{attribute 'linkalways'} 
{attribute 'no_explicit_call' := 'This FB is a CLASS and must be accessed using methods or properties'}
{attribute 'enable_dynamic_creation'}
FUNCTION_BLOCK Node_F_VN_PutText EXTENDS Node
VAR
    sText : _STRING('');
    ipDestImage : _ITcVnImage;
    nX : _UDINT(1);
    nY : _UDINT(1);
    eFontType : _ETcVnFontType(ETcVnFontType.TCVN_FT_HERSHEY_SIMPLEX);
    fFontScale : _LREAL(1.0);
    //aColor : _TcVnVector4_LREAL;
    hrPrev : _HRESULT(S_OK);
	hresult : _HRESULT(S_OK);
END_VAR

METHOD PUBLIC  Clone : I_Node
VAR
	pNode : POINTER TO Node_F_VN_PutText;
END_VAR
pNode := __NEW(Node_F_VN_PutText);
Clone := pNode^;
END_METHOD

METHOD FB_init : BOOL
VAR_INPUT
	bInitRetains : BOOL; // if TRUE, the retain variables are initialized (warm start / cold start)
	bInCopyCode : BOOL;  // if TRUE, the instance afterwards gets moved into the copy code (online change)
END_VAR
AddInput('sText', sText);
AddInput('ipDestImage', ipDestImage);
//AddInput('aColor', aColor);
AddInput('hrPrev', hrPrev);
AddOutput('ipDestImage', ipDestImage);
AddOutput('hresult',hresult);
AddParameter('nX', nX);
AddParameter('nY', nY);
AddParameter('eFontType', eFontType);
AddParameter('fFontScale', fFontScale);
END_METHOD

METHOD PROTECTED  OnExecute : HRESULT

//REMOVE
VAR
    aColor_Green : TcVnVector4_LREAL := [0, 255, 0];
END_VAR
hresult.Value := F_VN_PutText(
    sText := sText.Value,
	ipDestImage := ipDestImage.Value,
	nX:= nX.Value,
	nY:= nY.Value,
    eFontType := eFontType.Value,
    fFontScale := fFontScale.Value,
    //aColor := aColor.Value,
    aColor := aColor_Green,
	hrPrev:= hrPrev.Value);
END_METHOD

END_FUNCTION_BLOCK

(* stored: Version 1.1.0.1, ProductVersion 3.1.4024.13
   POU Node_F_VN_PutText: Id {dbb9b54a-920b-09ce-09c9-bd4922723564}, SpecialFunc None
   Folder Constructor: Id {f9149f9f-7d0d-0ca9-09ed-43ae7099623a}
   Method Clone: Id {6a37ce67-8e32-091e-0319-f3cb46f59737}
   Method FB_init: Id {d08bfaae-dec8-03bc-0cdc-1a00485cdea4}
   Method OnExecute: Id {a44f2922-7f9d-0a5f-0dfa-fd8ca1736e22} *)
